FUNCTION TFPackOnPickPoint : BOOL
VAR_INPUT
	WorkPickPointState : POINTER TO ARRAY [1..MAXPICKPOINT] OF TFMachinePalletizer_WorkPickPointState;
END_VAR
VAR
	wpp : INT;
END_VAR

TFPackOnPickPoint := FALSE;

FOR wpp:=1 TO MAXPICKPOINT DO
	(* Verifico disponibilità Pacco *)
	IF WorkPickPointState^[wpp].State = WORKPICKPOINT_PRODOTTO_PRESENTE THEN
		TFPackOnPickPoint := TRUE;
	END_IF
END_FOR

END_FUNCTION

(* stored: Version 1.1.0.1, ProductVersion 3.1.4024.11
   POU TFPackOnPickPoint: Id {1b4232c3-d445-43d2-ae79-174f0fad6996}, SpecialFunc None *)
